TEXTLIST TL_Busy
  0 = 'Begin Test'
  1 = 'Break Test'
   = ''
END_TEXTLIST

(* stored: Version 1.1.0.1, ProductVersion 3.1.4020.3
   TextList TL_Busy: Id {74b21f0b-9db1-4fb5-8ec0-31e87e50d72c} *)
